PROGRAM MAIN
VAR	
	// Timers
	Timer : TON;
	TimerOn : BOOL := FALSE;
END_VAR

Timer(IN := TimerOn, PT := T#30S); // Start de timer voor 30 seconden

// Case 1: Productdetectie (detecteer producten op de band en start de motor).
IF GVL.caseInput = 1 THEN // Controleer of het eerste product gedetecteerd is en het tweede niet
    GVL.MotorStatus := TRUE; // Zet de motorstatus aan (start de motor)
END_IF

// Case 2: Als de motor aan staat moet een timer gaan lopen die de tijd opneemt hoe lang de band loopt.
IF GVL.caseInput = 2 THEN
	TimerOn := TRUE; // Start de timer.
	IF Timer.ET > T#1S THEN // Controleer of de band langer als een seconde loopt
		GVL.ProductGedetecteerd1 := FALSE; // Zet de sensor productgedetecteerd uit
	END_IF
END_IF

// Case 3: Stoppen van de band (stop de motor na het bereiken van het einddoel).
IF GVL.caseInput = 3 THEN // Controleer of het tweede product gedetecteerd is en de band al langer als een seconde loopt
    IF GVL.MotorStatus THEN
		POU(Timer.ET); // Geef de afstand en tijd wat het object er over heeft gedaan mee aan de functie
	END_IF 
	GVL.MotorStatus := 0; // Zet de motorstatus uit (stop de motor)
	TimerOn := FALSE;
END_IF

END_PROGRAM

(* stored: Version 1.1.0.1, ProductVersion 3.1.4024.12
   POU MAIN: Id {cf05c820-487e-4dd3-a2e9-a0782d731133}, SpecialFunc None *)
